KUKA KRL program: Weld_PartB.src, Weld_PartB.dat

--- Weld_PartB.src ---
&ACCESS RVP
&REL 1
&COMMENT Han co xe Wave Alpha
DEF Weld_PartB()
  ;FOLD INI
    ;FOLD BASISTECH INI
      BAS(#INITMOV, 0)
    ;ENDFOLD
  ;ENDFOLD

  PTP HOME Vel=100% DEFAULT

  LIN P1
  LIN P2

  PTP HOME Vel=100% DEFAULT

END

--- Weld_PartB.dat ---
&ACCESS RV
&REL 1
DEFDAT Weld_PartB PUBLIC
  DECL E6POS HOME={A1 0.0, A2 -90.0, A3 90.0, A4 0.0, A5 0.0, A6 0.0}
  DECL E6POS P1={X 300.0, Y 0.0, Z 200.0, A 0.0, B 90.0, C 0.0, S 2, T 10}
  DECL E6POS P2={X 300.0, Y 150.0, Z 200.0, A 0.0, B 90.0, C 0.0, S 2, T 10}
ENDDAT
